Staubli VAL3: Form_4jHome.pgx

public program Form_4jHome(string x_sTitle, jointRs& x_jJ)
begin
  //call Form_MainS(",,,,,记录,保存,退出")
  title(x_sTitle)

  call Form_PattenS(x_sTitle,"记录,,,,,,保存,退出","记录,,,,,,保存,退出")
  call Control_PanelXY(22,0,15,10)
  call Control_Panel("Home")
  //call con
  gotoxy(nPanelLTopX+1,nPanelLTopY+1)
  put(left("j1:"+toString(".3",x_jJ.j1)+"        ",nPanelWidthX))

  gotoxy(nPanelLTopX+1,nPanelLTopY+2)
  put(left("j2:"+toString(".3",x_jJ.j2)+"        ",nPanelWidthX))

  gotoxy(nPanelLTopX+1,nPanelLTopY+3)
  put(left("j3:"+toString(".3",x_jJ.j3)+"        ",nPanelWidthX))

  gotoxy(nPanelLTopX+1,nPanelLTopY+4)
  put(left("j4:"+toString(".3",x_jJ.j4)+"        ",nPanelWidthX))



end
